Universal Robots PolyScope program: dominos-v1.urp

Program dominos-v1 (installation=default directory=/programs/usbdisk createdIn=5.12.2.1101534 lastSavedIn=5.12.2.1101534 robotSerialNumber=20225300872)
Calibrated DH parameters: a=[-0.000084, -0.221352, -0.21153, 0.000055, -0.000098, 0]; d=[0.151861, 36.284024, -28.917988, -7.234922, 0.085399, 0.092121]; alpha=[1.570877, 0.002818, 0.003813, 1.571803, -1.572963, 0]; deltaTheta=[0, 0.43274, -0.300741, -0.132009, 0.000003, 0]
Robot Program (runOnlyOnce=false)
  Folder Init main
    URCap Activer la main (Robotiq_Grippers, Robotiq Inc.) dataModel(ResetAndActivateKey=false)
    URCap Main (Robotiq_Grippers, Robotiq Inc.) dataModel(position=60.0, force=0.0, speed=0.0, positionInDouble=60.0, forceInDouble=0.0, speedInDouble=0.0, slaveIds=[9], blocking=true)
  Folder init vars
    offest_rx := 3.14
    topz := 0.280
    offset := 0.250
  MoveJ speed 60 deg/s, acceleration 80 deg/s^2 (useActiveTCP=true) feature=Base
    Waypoint start_pos: TCP in base x=172.583 y=-199.697 z=280.013 mm, rx=2.1282 ry=2.3108 rz=0 rad; joints [340.785, -73.502, -110.261, -86.109, 90.107, 155.995] deg; TCP offset x=0 y=0 z=0 mm, rx=0 ry=0 rz=0 rad
  Folder init prod
    URCap EYE+ Control (Asyril-EYE+, Asyril SA) dataModel(advancedMethodKey=false, command=stop, parameter=production, xmlrpc_s1KEY=XR_EYE_s1, xmlrpc_s2KEY=XR_EYE_s2, eyePlusName=EYE, title_key=EYE stop production, nodeDefined=true)
    URCap EYE+ Control (Asyril-EYE+, Asyril SA) dataModel(advancedMethodKey=false, command=start_production, parameter=4875, xmlrpc_s1KEY=XR_EYE_s1, xmlrpc_s2KEY=XR_EYE_s2, eyePlusName=EYE, title_key=EYE start_production 4875, nodeDefined=true)
    erreur_eye := EYECheckLastError()
    If erreur_eye≠0
      Popup Message (haltProgram=false inputType=Variable) variable=erreur_eye
      Halt
  Loop Forever
    Folder prod
      URCap EYE+ Control (Asyril-EYE+, Asyril SA) dataModel(advancedMethodKey=false, command=get_part, xmlrpc_s1KEY=XR_EYE_s1, xmlrpc_s2KEY=XR_EYE_s2, eyePlusName=EYE, title_key=EYE get_part, nodeDefined=true, Variable(key=EYEPos, variable(name=EYEPos, initializeExpression=p[0,0,0,0,0,0])))
      If EYEPos≟p[0,0,0,0,0,0]
        Halt
      EYEPos := pose_add(EYEPos,p[0,0,0,0,0,0])
      EYEPos := pose_add(EYEPos, p[0,0,0,offest_rx,0,0])
      EYEPosTop := pose_add(EYEPos, p[0,0,topz,0,0,0])
      EYEPosOffset := pose_add(EYEPos, p[0,0,offset,0,0,0])   [initializeExpression=p[0,0,0,0,0,0]]
      MoveJ speed 60 deg/s, acceleration 80 deg/s^2 (useActiveTCP=true) feature=Base
        Waypoint Waypoint (Variable): variable=EYEPosTop
        Waypoint Waypoint (Variable): variable=EYEPosOffset
      URCap Main (Robotiq_Grippers, Robotiq Inc.) dataModel(position=66.88235294117646, force=0.0, speed=0.0, positionInDouble=66.88235294117646, forceInDouble=0.0, speedInDouble=0.0, slaveIds=[9], blocking=true)
      MoveL speed 250 mm/s, acceleration 1200 mm/s^2 (useActiveTCP=true) feature=Base
        Waypoint Waypoint (Variable): variable=EYEPosTop
        Waypoint pos_boite: TCP in base x=-97.635 y=-349.696 z=279.997 mm, rx=2.2547 ry=2.1649 rz=-0.0119 rad; joints [275.65, -99.364, -86.669, -82.861, 90.392, 97.879] deg
      URCap Main (Robotiq_Grippers, Robotiq Inc.) dataModel(position=60.0, force=0.0, speed=0.0, positionInDouble=60.0, forceInDouble=0.0, speedInDouble=0.0, slaveIds=[9], blocking=true)
  URCap EYE+ Control (Asyril-EYE+, Asyril SA) dataModel(advancedMethodKey=false, command=stop, parameter=production, xmlrpc_s1KEY=XR_EYE_s1, xmlrpc_s2KEY=XR_EYE_s2, eyePlusName=EYE, title_key=EYE stop production, nodeDefined=true)
